PROGRAM MAIN
VAR
END_VAR

END_PROGRAM

(* stored: Version 1.1.0.1
   POU MAIN: Id {f5c4bcce-ee91-4d05-9f8b-5d73ff284572} *)
